FUNCTION_BLOCK E_TRIG (* Trigger unconnected input events of the specified type inside a resource *)
  (* Standard: 61499-1; Classification: Event-driven blocks; Function: Auto-Trigger Block; Description: Copyright (c) 2025 Mario Kastner, HR Agrartechnik GmbH This program and the accompanying materials are made available under the terms of the Eclipse Public License 2.0 which is available at https://www.eclipse.org/legal/epl-2.0/ SPDX-License-Identifier: EPL-2.0 *)
  (* Version 1.0, 2025-01-08, Mario Kastner *)
  (* Version 3.0, 2025-04-14, Franz Höpfinger, HR Agrartechnik GmbH, Made Version 3.0.0 inspired by Work from Patrick Aigner *)
  PACKAGE iec61499::events;
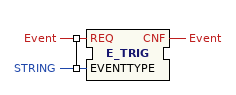
  EVENT_INPUT
    REQ WITH EVENTTYPE; (* Request trigger of unconnected event pins of type EVENTTYPE *)
  END_EVENT
  EVENT_OUTPUT
    CNF; (* Confirmation of Requested Service *)
  END_EVENT
  VAR_INPUT
    EVENTTYPE : STRING := 'EInit'; (* Event type to be triggered *)
  END_VAR
END_FUNCTION_BLOCK
